DATA_BLOCK "ST10_Flow27_KReserveLoad&Unload_iDB"
VAR
  sCtrlMode : "SysFlowCtrlGraph";
  sUpdMES_Data : Bool;
  "工件放行中" : Bool;
  "前站站号" : UInt;
  "本站站号" : UInt;
  "弹窗Temp" : Array[1..10] of Int;
  AlarmID : Int;
  TON : Array[0..10] of TON_TIME;
  TOF : Array[0..10] of TOF_TIME;
  sUP : Array[0..10] of Bool;
  "更新RFID完成" : Bool;
  RT_DATA : G7_RTDataPlus_V6;
  Trans1 : G7_TransitionPlus_V6;
  Trans2 : G7_TransitionPlus_V6;
  Trans3 : G7_TransitionPlus_V6;
  Trans102 : G7_TransitionPlus_V6;
  Trans28 : G7_TransitionPlus_V6;
  Trans29 : G7_TransitionPlus_V6;
  Trans30 : G7_TransitionPlus_V6;
  Trans31 : G7_TransitionPlus_V6;
  Trans32 : G7_TransitionPlus_V6;
  Trans33 : G7_TransitionPlus_V6;
  Trans34 : G7_TransitionPlus_V6;
  Trans35 : G7_TransitionPlus_V6;
  Trans36 : G7_TransitionPlus_V6;
  Trans37 : G7_TransitionPlus_V6;
  Trans38 : G7_TransitionPlus_V6;
  Trans39 : G7_TransitionPlus_V6;
  Trans40 : G7_TransitionPlus_V6;
  Trans41 : G7_TransitionPlus_V6;
  Trans42 : G7_TransitionPlus_V6;
  Trans43 : G7_TransitionPlus_V6;
  Trans44 : G7_TransitionPlus_V6;
  Trans45 : G7_TransitionPlus_V6;
  Trans46 : G7_TransitionPlus_V6;
  Trans47 : G7_TransitionPlus_V6;
  Trans48 : G7_TransitionPlus_V6;
  Trans49 : G7_TransitionPlus_V6;
  Trans50 : G7_TransitionPlus_V6;
  Trans51 : G7_TransitionPlus_V6;
  Trans52 : G7_TransitionPlus_V6;
  Trans53 : G7_TransitionPlus_V6;
  Trans54 : G7_TransitionPlus_V6;
  Trans55 : G7_TransitionPlus_V6;
  Trans56 : G7_TransitionPlus_V6;
  Trans57 : G7_TransitionPlus_V6;
  Trans58 : G7_TransitionPlus_V6;
  Trans59 : G7_TransitionPlus_V6;
  Trans60 : G7_TransitionPlus_V6;
  Trans61 : G7_TransitionPlus_V6;
  Trans62 : G7_TransitionPlus_V6;
  Trans63 : G7_TransitionPlus_V6;
  Trans64 : G7_TransitionPlus_V6;
  Trans65 : G7_TransitionPlus_V6;
  Trans66 : G7_TransitionPlus_V6;
  Trans67 : G7_TransitionPlus_V6;
  Trans68 : G7_TransitionPlus_V6;
  Trans69 : G7_TransitionPlus_V6;
  Trans70 : G7_TransitionPlus_V6;
  Trans71 : G7_TransitionPlus_V6;
  Trans72 : G7_TransitionPlus_V6;
  Trans73 : G7_TransitionPlus_V6;
  Trans74 : G7_TransitionPlus_V6;
  Trans75 : G7_TransitionPlus_V6;
  Trans76 : G7_TransitionPlus_V6;
  Trans77 : G7_TransitionPlus_V6;
  Trans78 : G7_TransitionPlus_V6;
  Trans79 : G7_TransitionPlus_V6;
  Trans80 : G7_TransitionPlus_V6;
  Trans81 : G7_TransitionPlus_V6;
  Trans82 : G7_TransitionPlus_V6;
  Trans200 : G7_TransitionPlus_V6;
  Trans765 : G7_TransitionPlus_V6;
  Trans766 : G7_TransitionPlus_V6;
  Trans767 : G7_TransitionPlus_V6;
  Trans119 : G7_TransitionPlus_V6;
  Trans120 : G7_TransitionPlus_V6;
  Trans121 : G7_TransitionPlus_V6;
  Trans122 : G7_TransitionPlus_V6;
  Trans123 : G7_TransitionPlus_V6;
  Trans768 : G7_TransitionPlus_V6;
  Trans769 : G7_TransitionPlus_V6;
  Trans126 : G7_TransitionPlus_V6;
  Trans127 : G7_TransitionPlus_V6;
  Trans128 : G7_TransitionPlus_V6;
  Trans124 : G7_TransitionPlus_V6;
  Trans770 : G7_TransitionPlus_V6;
  Trans771 : G7_TransitionPlus_V6;
  Trans129 : G7_TransitionPlus_V6;
  Trans130 : G7_TransitionPlus_V6;
  Trans131 : G7_TransitionPlus_V6;
  Trans125 : G7_TransitionPlus_V6;
  Trans132 : G7_TransitionPlus_V6;
  Trans772 : G7_TransitionPlus_V6;
  Trans773 : G7_TransitionPlus_V6;
  Trans133 : G7_TransitionPlus_V6;
  Trans134 : G7_TransitionPlus_V6;
  Trans776 : G7_TransitionPlus_V6;
  Trans142 : G7_TransitionPlus_V6;
  Trans143 : G7_TransitionPlus_V6;
  Trans135 : G7_TransitionPlus_V6;
  Trans136 : G7_TransitionPlus_V6;
  Trans774 : G7_TransitionPlus_V6;
  Trans775 : G7_TransitionPlus_V6;
  Trans137 : G7_TransitionPlus_V6;
  Trans138 : G7_TransitionPlus_V6;
  Trans139 : G7_TransitionPlus_V6;
  Trans140 : G7_TransitionPlus_V6;
  Trans777 : G7_TransitionPlus_V6;
  Trans778 : G7_TransitionPlus_V6;
  Trans141 : G7_TransitionPlus_V6;
  Trans144 : G7_TransitionPlus_V6;
  Trans146 : G7_TransitionPlus_V6;
  Trans147 : G7_TransitionPlus_V6;
  Trans779 : G7_TransitionPlus_V6;
  Trans780 : G7_TransitionPlus_V6;
  Trans148 : G7_TransitionPlus_V6;
  Trans149 : G7_TransitionPlus_V6;
  Trans150 : G7_TransitionPlus_V6;
  Trans163 : G7_TransitionPlus_V6;
  Trans164 : G7_TransitionPlus_V6;
  Trans165 : G7_TransitionPlus_V6;
  Trans166 : G7_TransitionPlus_V6;
  Trans167 : G7_TransitionPlus_V6;
  Trans151 : G7_TransitionPlus_V6;
  Trans152 : G7_TransitionPlus_V6;
  Trans153 : G7_TransitionPlus_V6;
  Trans168 : G7_TransitionPlus_V6;
  Trans781 : G7_TransitionPlus_V6;
  Trans782 : G7_TransitionPlus_V6;
  Trans783 : G7_TransitionPlus_V6;
  Trans154 : G7_TransitionPlus_V6;
  Trans155 : G7_TransitionPlus_V6;
  Trans784 : G7_TransitionPlus_V6;
  Trans785 : G7_TransitionPlus_V6;
  Trans156 : G7_TransitionPlus_V6;
  Trans157 : G7_TransitionPlus_V6;
  Trans158 : G7_TransitionPlus_V6;
  Trans159 : G7_TransitionPlus_V6;
  Trans786 : G7_TransitionPlus_V6;
  Trans787 : G7_TransitionPlus_V6;
  Trans160 : G7_TransitionPlus_V6;
  Trans161 : G7_TransitionPlus_V6;
  Trans162 : G7_TransitionPlus_V6;
  Trans169 : G7_TransitionPlus_V6;
  Trans788 : G7_TransitionPlus_V6;
  Trans789 : G7_TransitionPlus_V6;
  Trans170 : G7_TransitionPlus_V6;
  Trans171 : G7_TransitionPlus_V6;
  Trans172 : G7_TransitionPlus_V6;
  Trans173 : G7_TransitionPlus_V6;
  Trans174 : G7_TransitionPlus_V6;
  Trans175 : G7_TransitionPlus_V6;
  Trans197 : G7_TransitionPlus_V6;
  Trans198 : G7_TransitionPlus_V6;
  Trans176 : G7_TransitionPlus_V6;
  Trans145 : G7_TransitionPlus_V6;
  Trans177 : G7_TransitionPlus_V6;
  Trans202 : G7_TransitionPlus_V6;
  Trans203 : G7_TransitionPlus_V6;
  Trans204 : G7_TransitionPlus_V6;
  Trans205 : G7_TransitionPlus_V6;
  Trans206 : G7_TransitionPlus_V6;
  Trans207 : G7_TransitionPlus_V6;
  Trans250 : G7_TransitionPlus_V6;
  Trans251 : G7_TransitionPlus_V6;
  Trans252 : G7_TransitionPlus_V6;
  Trans253 : G7_TransitionPlus_V6;
  Trans254 : G7_TransitionPlus_V6;
  Trans255 : G7_TransitionPlus_V6;
  Trans256 : G7_TransitionPlus_V6;
  Trans257 : G7_TransitionPlus_V6;
  Trans258 : G7_TransitionPlus_V6;
  Trans259 : G7_TransitionPlus_V6;
  Trans260 : G7_TransitionPlus_V6;
  Trans613 : G7_TransitionPlus_V6;
  F27_Initial : G7_StepPlus_V6;
  S2 : G7_StepPlus_V6;
  S3 : G7_StepPlus_V6;
  S4 : G7_StepPlus_V6;
  S10_InitialFinish : G7_StepPlus_V6;
  MotorCWStart : G7_StepPlus_V6;
  MotorCWStart_1 : G7_StepPlus_V6;
  MotorRunDelay : G7_StepPlus_V6;
  MotorRunDelay_1 : G7_StepPlus_V6;
  StopProcess : G7_StepPlus_V6;
  LoadingStop_2 : G7_StepPlus_V6;
  LoadingStop_3 : G7_StepPlus_V6;
  LoadingStop_4 : G7_StepPlus_V6;
  CheckPalletExist : G7_StepPlus_V6;
  CheckPalletExist_1 : G7_StepPlus_V6;
  CheckMaterialDoorLock : G7_StepPlus_V6;
  MotorRun : G7_StepPlus_V6;
  WaitLineMotorReady : G7_StepPlus_V6;
  WaitPalletRequestRelease : G7_StepPlus_V6;
  WaitPalletArrveNextPos : G7_StepPlus_V6;
  WaitLineMotorReady_1 : G7_StepPlus_V6;
  WaitPalletRequestRelease_1 : G7_StepPlus_V6;
  WaitPalletArrveNextPos_1 : G7_StepPlus_V6;
  CheckPalletExist_2 : G7_StepPlus_V6;
  WaitLineMotorReady_2 : G7_StepPlus_V6;
  WaitPalletRequestRelease_2 : G7_StepPlus_V6;
  WaitPalletArrveNextPos_2 : G7_StepPlus_V6;
  CheckPalletExist_3 : G7_StepPlus_V6;
  WaitLineMotorReady_3 : G7_StepPlus_V6;
  WaitPalletRequestRelease_3 : G7_StepPlus_V6;
  WaitPalletArrveNextPos_3 : G7_StepPlus_V6;
  CheckPalletExist_4 : G7_StepPlus_V6;
  WaitLineMotorReady_4 : G7_StepPlus_V6;
  WaitPalletRequestRelease_4 : G7_StepPlus_V6;
  WaitPalletArrveNextPos_4 : G7_StepPlus_V6;
  CheckPalletExist_5 : G7_StepPlus_V6;
  WaitLineMotorReady_5 : G7_StepPlus_V6;
  WaitPalletRequestRelease_5 : G7_StepPlus_V6;
  WaitPalletArrveNextPos_5 : G7_StepPlus_V6;
  CheckPalletExist_6 : G7_StepPlus_V6;
  WaitLineMotorReady_6 : G7_StepPlus_V6;
  WaitPalletRequestRelease_6 : G7_StepPlus_V6;
  WaitPalletArrveNextPos_6 : G7_StepPlus_V6;
  LoadStop_14 : G7_StepPlus_V6;
  LoadStop_12 : G7_StepPlus_V6;
  LoadStop_13 : G7_StepPlus_V6;
  CheckPalletExist_7 : G7_StepPlus_V6;
  WaitLineMotorReady_7 : G7_StepPlus_V6;
  WaitPalletRequestRelease_7 : G7_StepPlus_V6;
  WaitPalletArrveNextPos_7 : G7_StepPlus_V6;
  CheckPalletExist_8 : G7_StepPlus_V6;
  WaitLineMotorReady_8 : G7_StepPlus_V6;
  WaitPalletRequestRelease_8 : G7_StepPlus_V6;
  WaitPalletArrveNextPos_8 : G7_StepPlus_V6;
  CheckPalletExist_9 : G7_StepPlus_V6;
  WaitLineMotorReady_9 : G7_StepPlus_V6;
  WaitPalletRequestRelease_9 : G7_StepPlus_V6;
  WaitPalletArrveNextPos_9 : G7_StepPlus_V6;
  CheckPalletExist_10 : G7_StepPlus_V6;
  WaitLineMotorReady_10 : G7_StepPlus_V6;
  WaitPalletRequestRelease_10 : G7_StepPlus_V6;
  WaitPalletArrveNextPos_10 : G7_StepPlus_V6;
  MotorRun_1 : G7_StepPlus_V6;
  "MiddleNoPallet?" : G7_StepPlus_V6;
  ProcessStart : G7_StepPlus_V6;
  StoperReset : G7_StepPlus_V6;
  StoperReset_1 : G7_StepPlus_V6;
  StoperRelease_1 : G7_StepPlus_V6;
  AriveTimeDelay_1 : G7_StepPlus_V6;
  AriveTimeDelay_2 : G7_StepPlus_V6;
  StoperReset_2 : G7_StepPlus_V6;
  StoperRelease_2 : G7_StepPlus_V6;
  WaitPalletArive : G7_StepPlus_V6;
  TimeDelay : G7_StepPlus_V6;
  AriveTimeDelay_3 : G7_StepPlus_V6;
  StoperReset_3 : G7_StepPlus_V6;
  StoperRelease_3 : G7_StepPlus_V6;
  WaitPalletArive_1 : G7_StepPlus_V6;
  TimeDelay_1 : G7_StepPlus_V6;
  AriveTimeDelay_4 : G7_StepPlus_V6;
  StoperReset_4 : G7_StepPlus_V6;
  MotorStop : G7_StepPlus_V6;
  StoperRelease_4 : G7_StepPlus_V6;
  WaitPalletArive_2 : G7_StepPlus_V6;
  TimeDelay_2 : G7_StepPlus_V6;
  AriveTimeDelay_5 : G7_StepPlus_V6;
  StoperReset_5 : G7_StepPlus_V6;
  StoperRelease_5 : G7_StepPlus_V6;
  WaitPalletArive_3 : G7_StepPlus_V6;
  TimeDelay_3 : G7_StepPlus_V6;
  AriveTimeDelay_6 : G7_StepPlus_V6;
  LoadingStop_1 : G7_StepPlus_V6;
  Step143 : G7_StepPlus_V6;
  StoperReset_6 : G7_StepPlus_V6;
  StoperRelease_6 : G7_StepPlus_V6;
  WaitPalletArive_4 : G7_StepPlus_V6;
  TimeDelay_4 : G7_StepPlus_V6;
  AriveTimeDelay_7 : G7_StepPlus_V6;
  StoperReset_7 : G7_StepPlus_V6;
  StoperRelease_7 : G7_StepPlus_V6;
  WaitPalletArive_5 : G7_StepPlus_V6;
  TimeDelay_5 : G7_StepPlus_V6;
  Step153 : G7_StepPlus_V6;
  "CheckMachine Mode_1" : G7_StepPlus_V6;
  "CheckMachine Mode_2" : G7_StepPlus_V6;
  "CheckMachine Mode_3" : G7_StepPlus_V6;
  "CheckMachine Mode_4" : G7_StepPlus_V6;
  "CheckMachine Mode_5" : G7_StepPlus_V6;
  AriveTimeDelay_8 : G7_StepPlus_V6;
  LoadStop_11 : G7_StepPlus_V6;
  StoperReset_8 : G7_StepPlus_V6;
  StoperRelease_8 : G7_StepPlus_V6;
  AriveTimeDelay_9 : G7_StepPlus_V6;
  StoperReset_9 : G7_StepPlus_V6;
  StoperRelease_9 : G7_StepPlus_V6;
  WaitPalletArive_6 : G7_StepPlus_V6;
  TimeDelay_6 : G7_StepPlus_V6;
  AriveTimeDelay_10 : G7_StepPlus_V6;
  StoperReset_10 : G7_StepPlus_V6;
  StoperRelease_10 : G7_StepPlus_V6;
  WaitPalletArive_7 : G7_StepPlus_V6;
  TimeDelay_7 : G7_StepPlus_V6;
  AriveTimeDelay_11 : G7_StepPlus_V6;
  StoperReset_11 : G7_StepPlus_V6;
  StoperRelease_11 : G7_StepPlus_V6;
  WaitPalletArive_8 : G7_StepPlus_V6;
  TimeDelay_8 : G7_StepPlus_V6;
  "CheckMachine Mode_6" : G7_StepPlus_V6;
  "CheckMachine Mode_7" : G7_StepPlus_V6;
  "CheckMachine Mode_8" : G7_StepPlus_V6;
  WaitAllStoperReset : G7_StepPlus_V6;
  Step182 : G7_StepPlus_V6;
  WaitPalletArive_9 : G7_StepPlus_V6;
  TimeDelay_9 : G7_StepPlus_V6;
  CheckMachineMode : G7_StepPlus_V6;
  UnloadStoper_1 : G7_StepPlus_V6;
  UnloadStoper_2 : G7_StepPlus_V6;
  UnloadStoper_3 : G7_StepPlus_V6;
  "Process Finish_1" : G7_StepPlus_V6;
  "Process Finish_2" : G7_StepPlus_V6;
  "Process Finish_3" : G7_StepPlus_V6;
  "Process Finish_4" : G7_StepPlus_V6;
  "Process Finish_5" : G7_StepPlus_V6;
  "Process Finish_6" : G7_StepPlus_V6;
  "Process Finish_7" : G7_StepPlus_V6;
  "Process Finish_8" : G7_StepPlus_V6;
  "Process Finish_9" : G7_StepPlus_V6;
  "Process Finish_10" : G7_StepPlus_V6;
  "Process Finish_11" : G7_StepPlus_V6;
END_VAR
BEGIN
END_DATA_BLOCK
